FUNCTION_BLOCK FB_Panel EXTENDS FB_LinkDataDWord
VAR_INPUT
	nControlData  			: DWORD;
END_VAR

VAR_OUTPUT	
	nStatusData  			: DWORD;
END_VAR

SUPER^();
ControlData := nControlData;
nStatusData := StatusData;

END_FUNCTION_BLOCK

(* stored: Version 1.1.0.1, ProductVersion 3.1.4024.12
   POU FB_Panel: Id {e6254a7d-4ca8-06bd-1449-ca9d97b68dce}, SpecialFunc None *)
